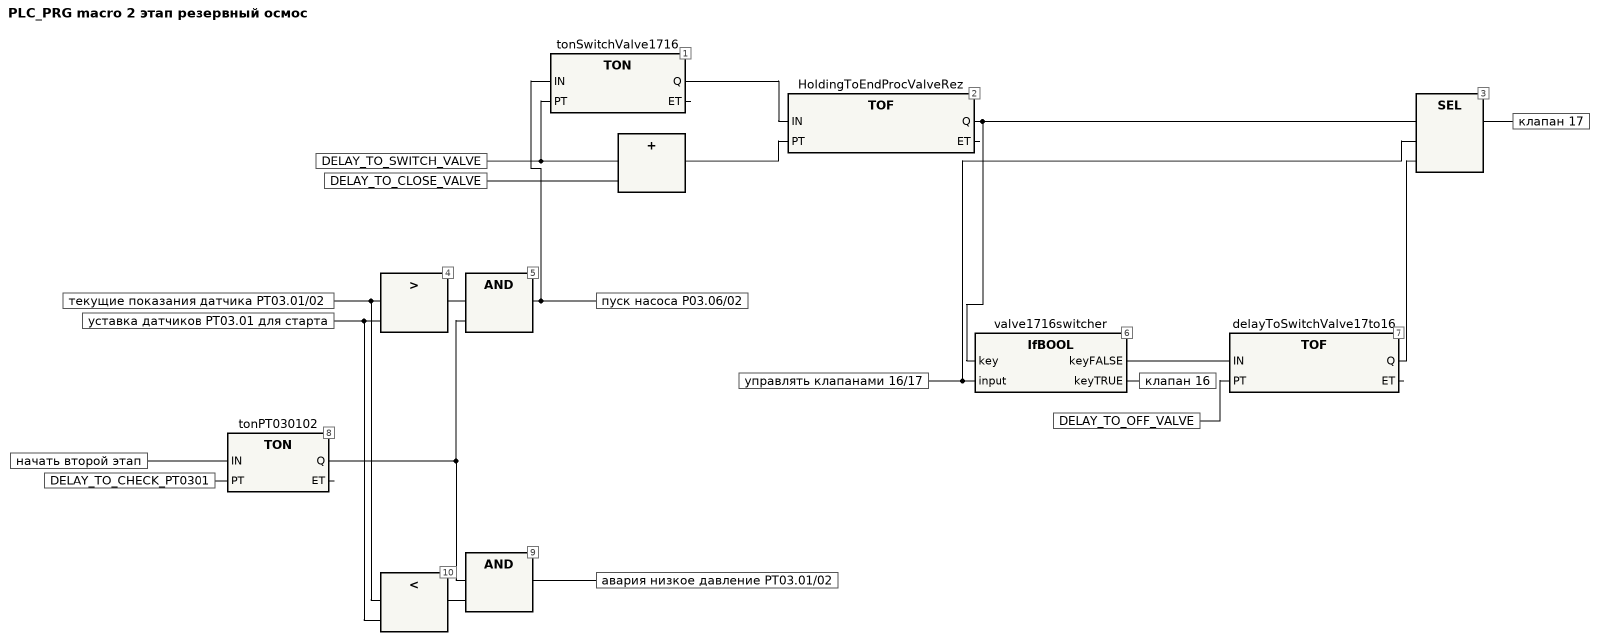
[picture p24: PLC_PRG macro 2 этап резервный осмос (CFC)]
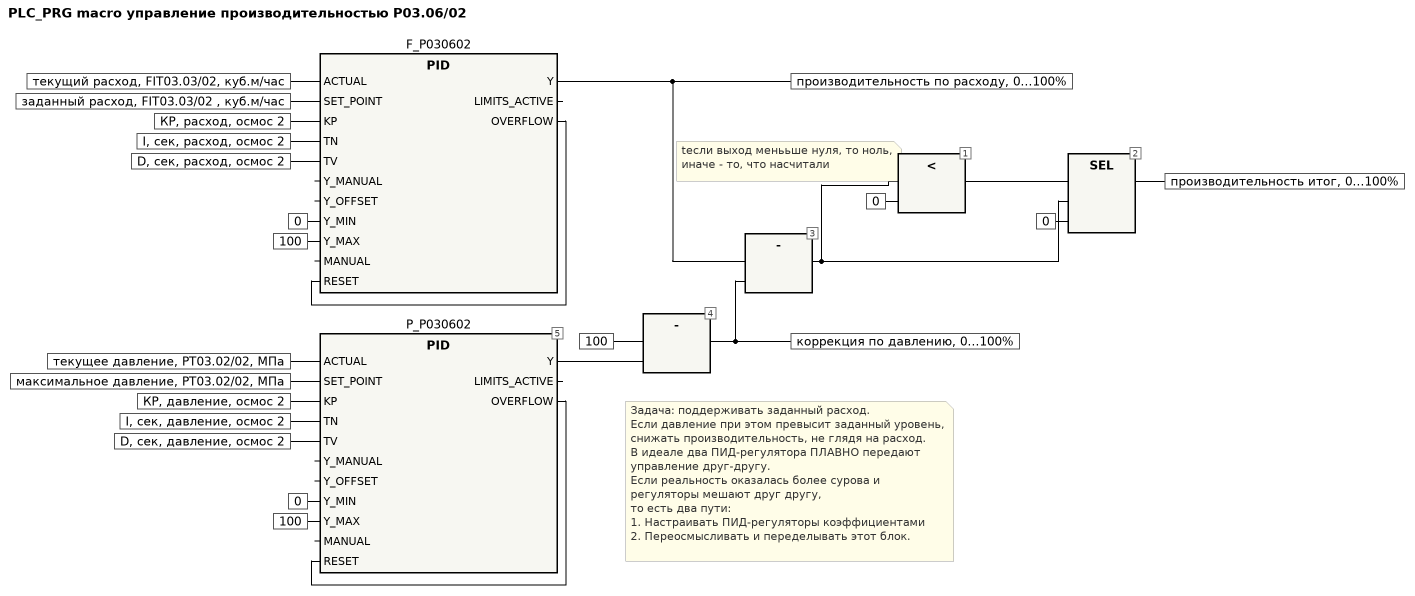
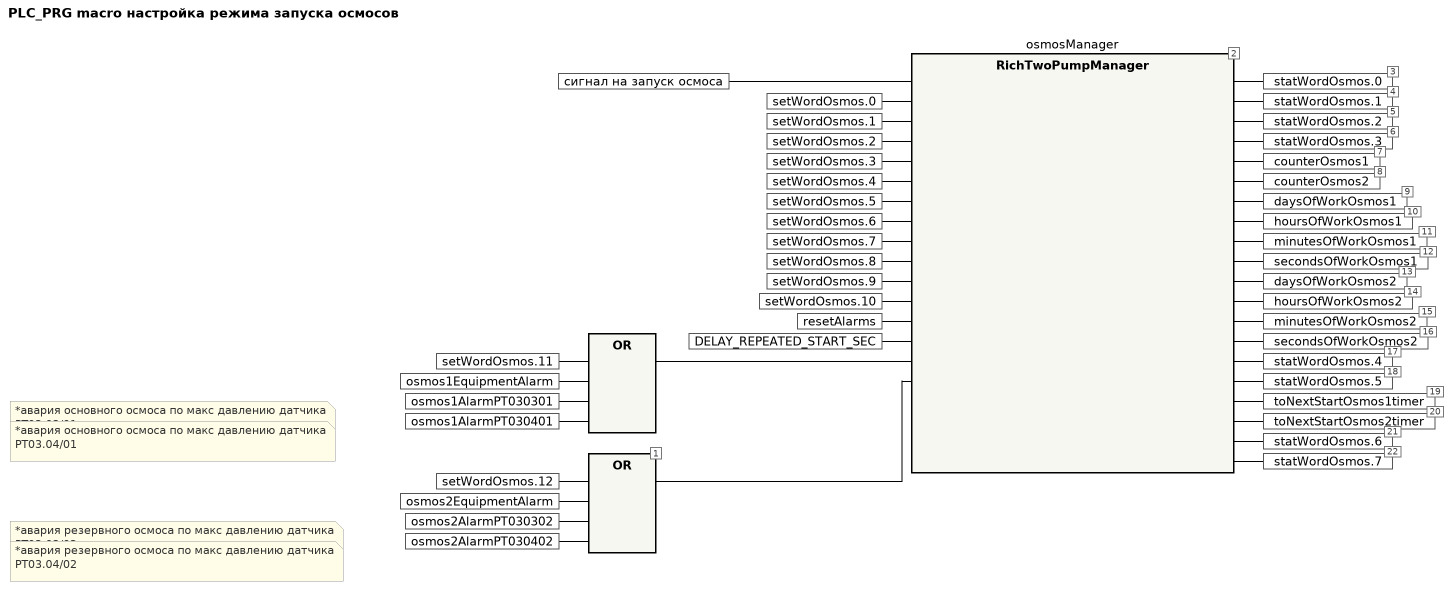
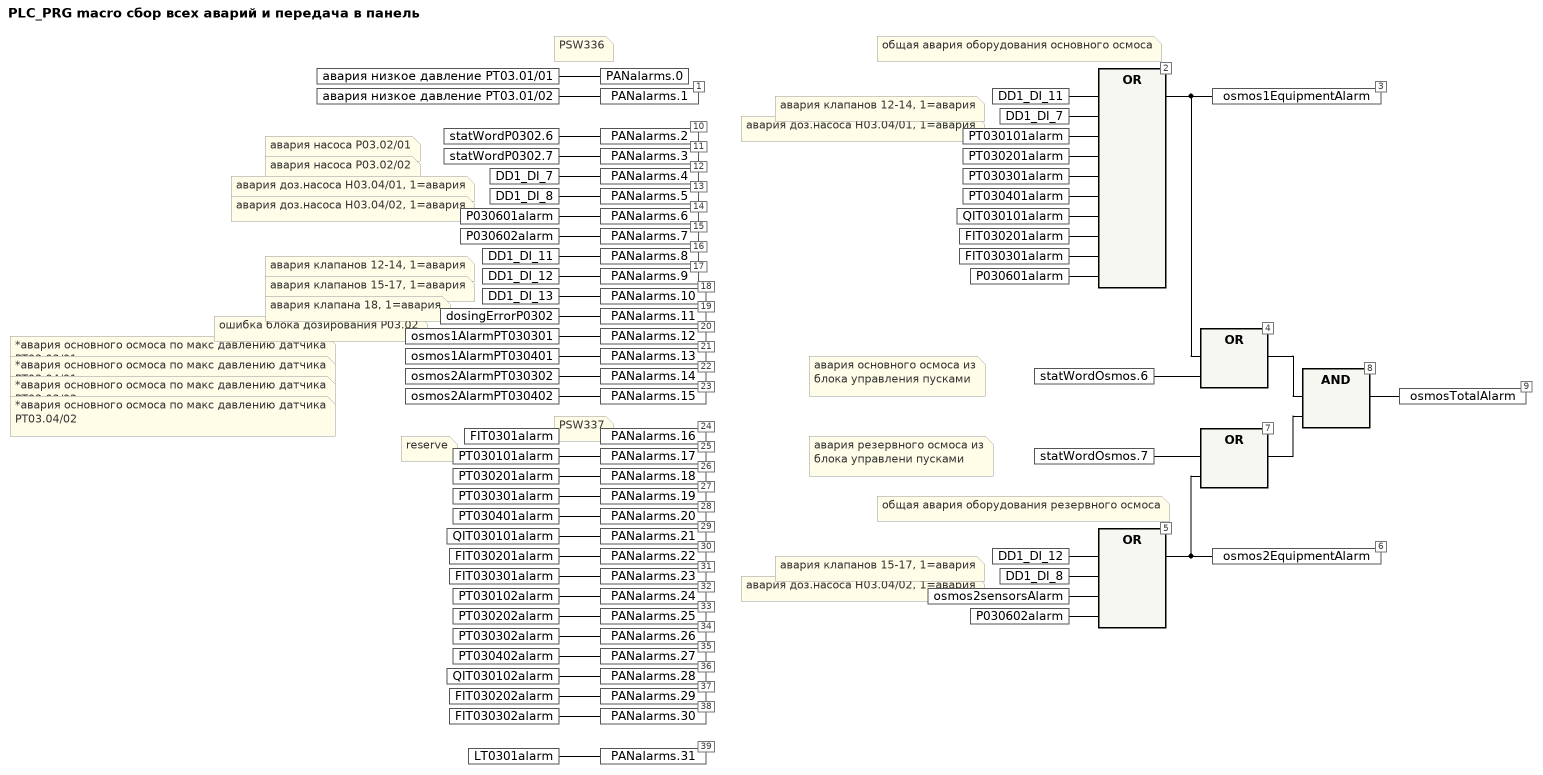
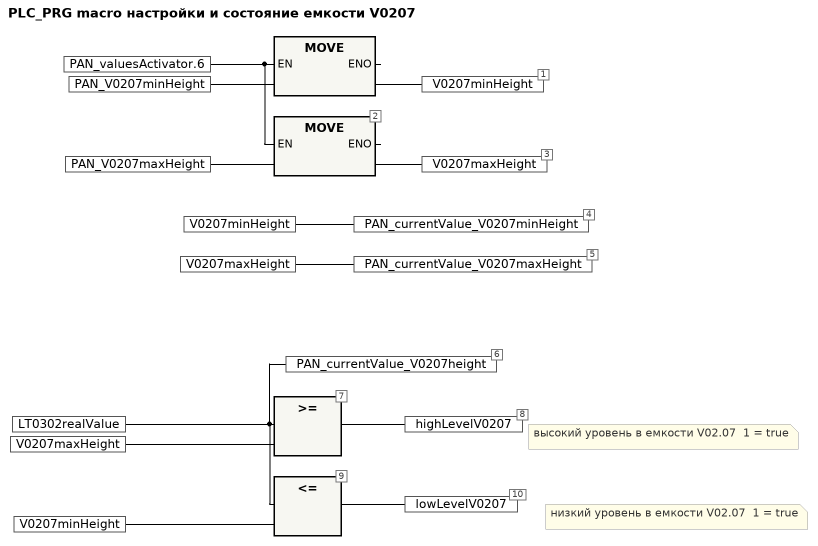
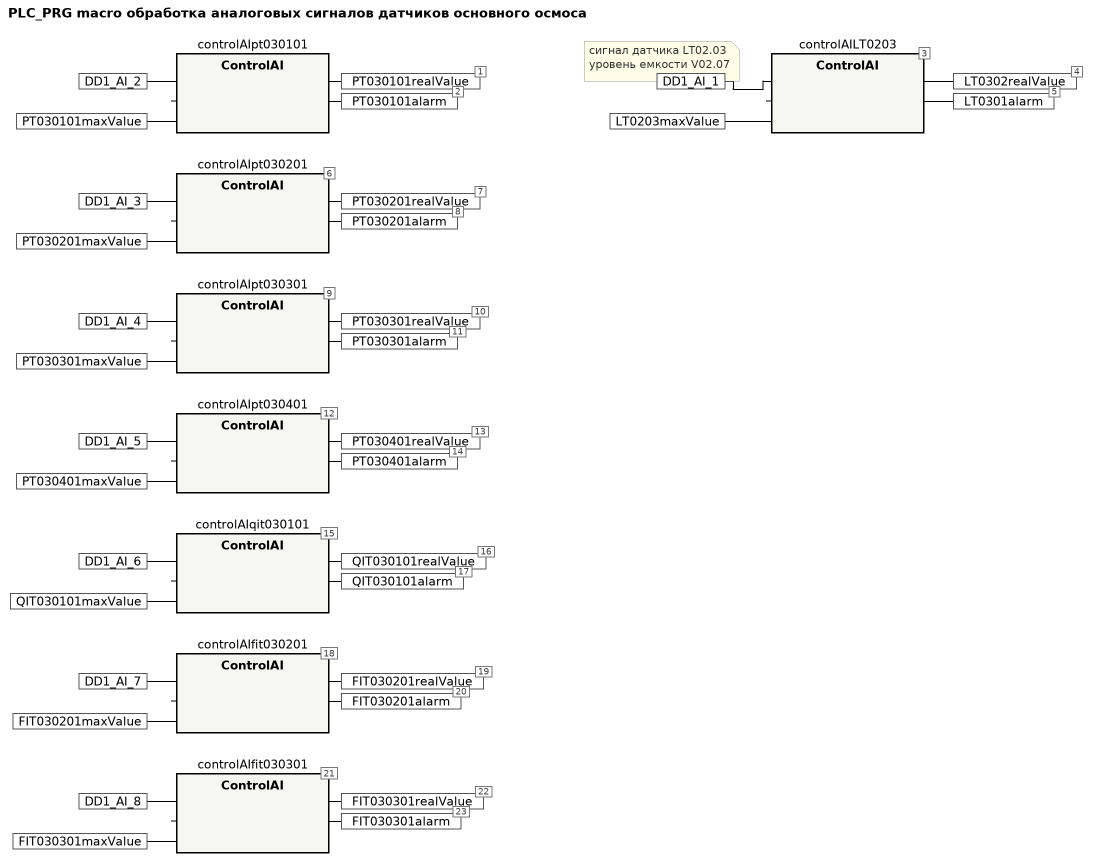
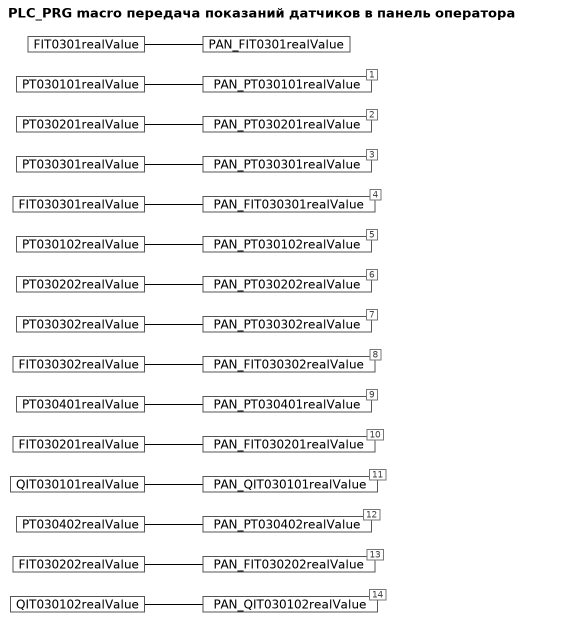
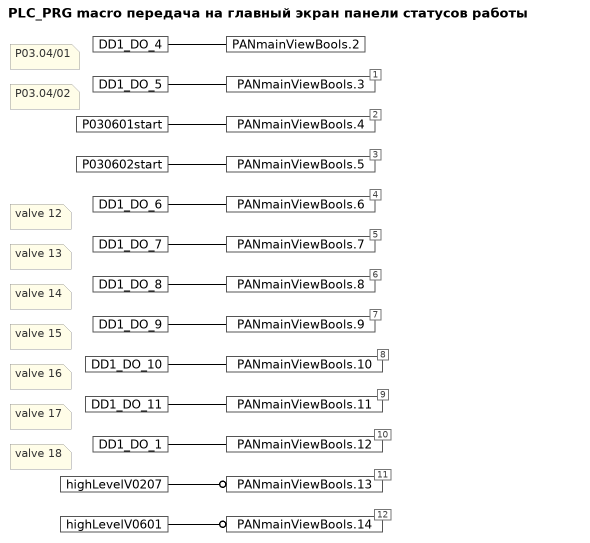
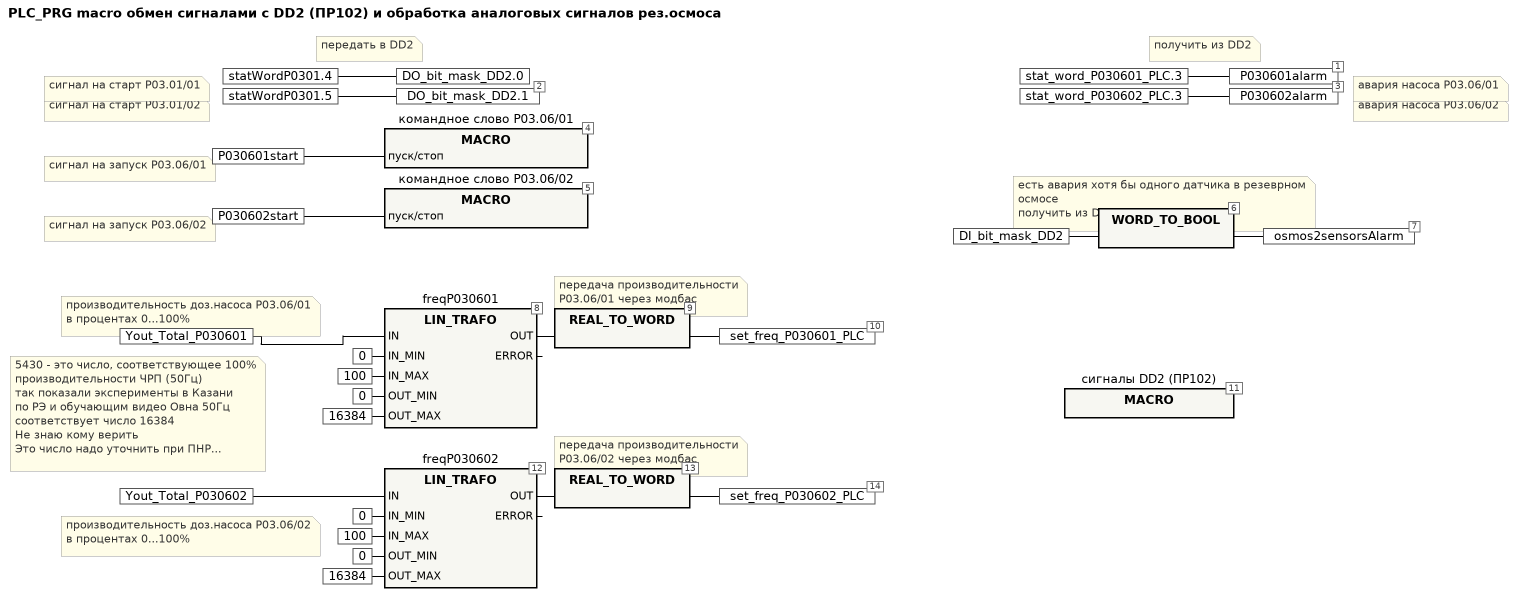
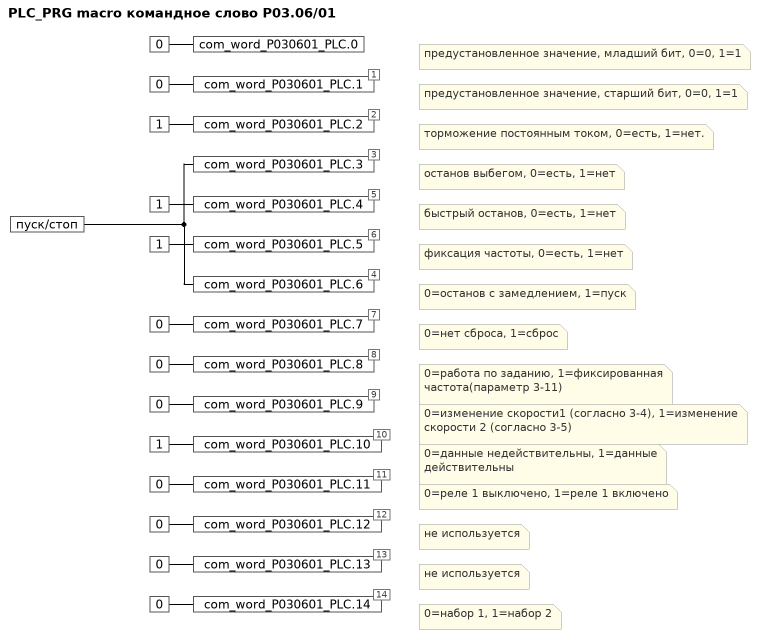
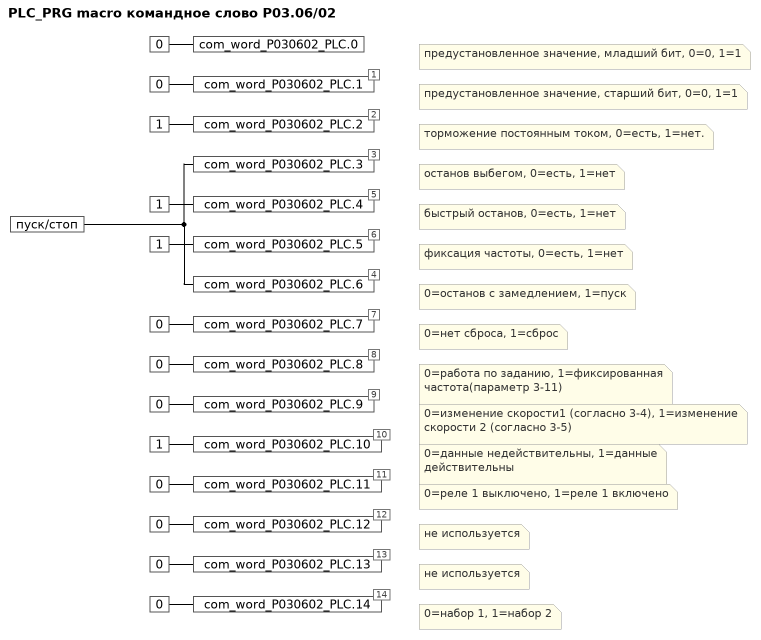
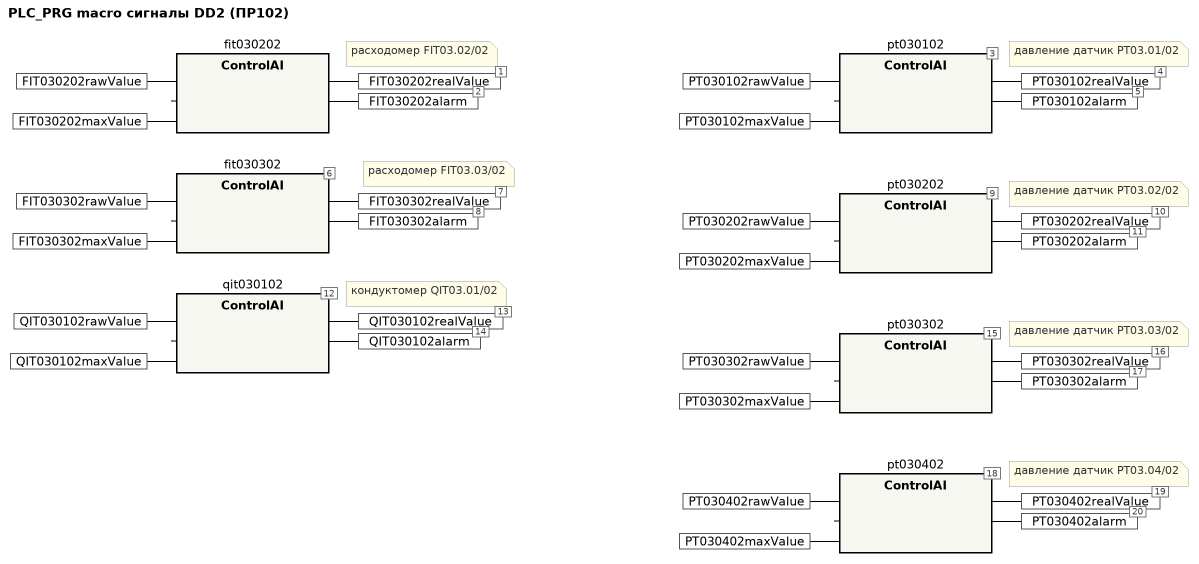
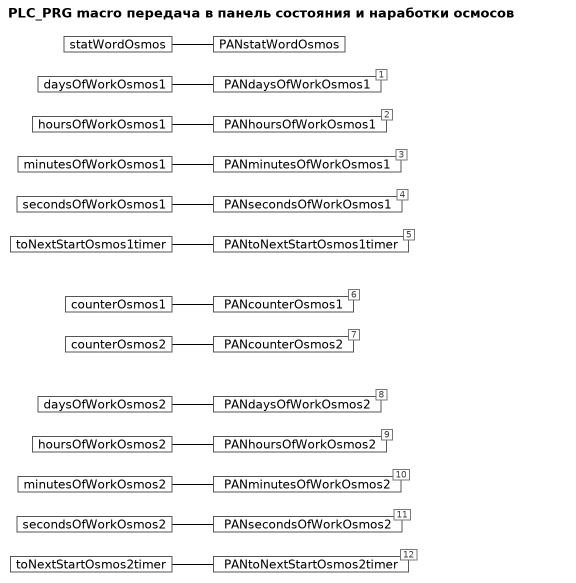
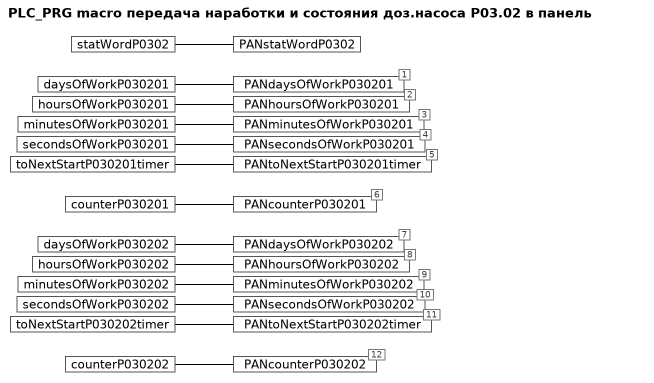
_CFC_ (* Continuous Function Chart, elements in execution order *)
(* принять сигнал из АСУ1, / FIT01.02, куб.м.час *)
(* Здесь это FIt01.02 / FIT0301 - название из алгоритма от второго осмоса *)
(* в осмосе 2 это было "Показания расходомера FIT03.01/01 на входе в осмос 2. / Для управления производительностью НД Р03.02 (1 и 2)." *)
(* пропиши в конфигурации ПЛК / ********************************** *)
(* пропиши в конфигурации ПЛК / ********************************** *)
(* авария обоих осмосов, 1 = авария *)
(* авария клапана 18, 1 = авария *)
(* авария обоих доз. насосов / Р03.02 на входе в осмос, 1 = авария *)
(* условие на запуск осмоса: / - высокий уровень в емкости V02.07 = false / - высокий уровень в емкости V06.01 = false / - высокий уровень в емкости V04.01 (БМТ) *)
(* - высокий уровень в емкости V02.07 / 1 = true *)
(* - высокий уровень в емкости V06.01 / (сигнал из АСУ-1 общий) 1 = true *)
(* алгоритм полностью скопирован из осмос-2 АСУ-3, / поэтому имена переменных многие будут оттуда, однако, в панели они / будут подписаны правильно! / Также здесь удалены насосы подачи на осмос Р03.01 / И условие запуска осмосов не такое, как в осмос-2 / Здесь запуск если V02.07  - !! нет сигнала что уровень высокий !! / (в осмос 2 - если уровень низкий) / емкость в БМТ не отслеживаем, а уровень в V06.01  условие то же / что и в осмос 2. *)
(* восстановление заданного ранее режима / работы после подачи питания *)
(* - высокий уровень в емкости V06.01 / (сигнал из АСУ-1 общий) 1 = true *)
(* расход в БМТ для расчета каскадной уставки / получить из АСУ-1! *)
(* показ расхода БМТ в панели оператора *)
(* 0 = уставка расходу своя, не каскад / 1 = уставка каскадная от расхода БМТ *)
(* прием/передача сигналов *)
(* командное слово для осмоса *)
(* командное слово доз. насоса Р03.02 *)
(* PAN - переменные для панели в щите / OPAN - переменные для выносной панели, на установке *)
(* ******************добавь сюда вкл и выкл от выносной панели******************* / задание режима работы - каскад/не каскад *)
(* передать в АСУ 1 для / передачи в осмос 2 *)
(* авария датчика уровня LT0203 *)
#0 onStartCatcher:R_TRIG(CLK: TRUE)
#1 OR(PANsetWordOsmos.11, #0.Q)
#2 resetAlarms <= #1
#3 setCascadeOnStart:IfBOOL(key: isCascadeOnStart, input: #0.Q)
#4 OR(#3.keyTRUE, PANsetWordOsmos.12)
#5 OR(#3.keyFALSE, PANsetWordOsmos.13)
#6 cascadeTrig:RS(SET: #4, RESET1: #5)
#7 statWordOsmos.8 <= #6.Q1
#8 isCascade <= #6.Q1
#9 OR(#4, #5)
#10 MOVE(EN: #9, isCascade)
#11 isCascadeOnStart <= #10
#12 MOVE(EN: #0.Q, setWordP0302onStart)
#13 setWordP0302 <= #12
#14 MOVE(EN: #0.Q, setWordOsmosOnStart)
#15 setWordOsmos <= #14
#16 ASU_Levels_output.0 <= lowLevelV0207
#17 highLevelV0601 <= ASU_Levels_input.0
#18 BMTflowToCascade <= ASU_FlowFromBMT
#19 FIT0301realValue <= ASU_FlowFIT0102
#20 MACRO алгоритм работы доз.насосов Р03.02(pin 1 "показания расходомера на входе": ASU_FlowFIT0102)
	(* приходит из макроса "алгоритм работы осмосов" *)
	(* авт.выкл и сигнал от самого / доз.насоса Р03.02/02 / 1 = норма, 0 = авария *)
	(* авт.выкл и сигнал от самого / доз.насоса Р03.02/01 / 1 = норма, 0 = авария *)
	(* Доз.насосы Р03.02/01 и Р03.02/02 на входе в осмос 2 *)
	(* выход на пуск Р03.02/01 *)
	(* задание производительности Р03.02/01 *)
	(* задание производительности Р03.02/02 *)
	(* выход на пуск Р03.02/02 *)
	(* invers alarms!!!!!!!!! *)
	#21 P0302:RichTwoPumpManager(startP0302, setWordP0302.0, setWordP0302.1, setWordP0302.2, setWordP0302.3, setWordP0302.4, setWordP0302.5, setWordP0302.6, setWordP0302.7, setWordP0302.8, setWordP0302.9, setWordP0302.10, resetAlarms, DELAY_REPEATED_START_SEC, DD1_DI_5, DD1_DI_6)
	#22 statWordP0302.0 <= #21.out 1
	#23 statWordP0302.1 <= #21.out 2
	#24 statWordP0302.2 <= #21.out 3
	#25 statWordP0302.3 <= #21.out 4
	#26 counterP030201 <= #21.out 5
	#27 counterP030202 <= #21.out 6
	#28 daysOfWorkP030201 <= #21.out 7
	#29 hoursOfWorkP030201 <= #21.out 8
	#30 minutesOfWorkP030201 <= #21.out 9
	#31 secondsOfWorkP030201 <= #21.out 10
	#32 daysOfWorkP030202 <= #21.out 11
	#33 hoursOfWorkP030202 <= #21.out 12
	#34 minutesOfWorkP030202 <= #21.out 13
	#35 secondsOfWorkP030202 <= #21.out 14
	#36 statWordP0302.4 <= #21.out 15
	#37 DD1_DO_2 <= #21.out 15
	#38 DD1_DO_3 <= #21.out 16
	#39 toNextStartP030201timer <= #21.out 17
	#40 statWordP0302.5 <= #21.out 16
	#41 toNextStartP030202timer <= #21.out 18
	#42 statWordP0302.6 <= #21.out 19
	#43 statWordP0302.7 <= #21.out 20
	#44 SEL(statWordP0302.4, 4.00, #46.out 1)
	#45 DD1_AO_1 <= #44
	#46 P0302dos:DosingPumpProportional(pin 1, -, setMaxPumpDosingValueP0302, -, -, setKoeffProportionalityP0302, -)
	#47 dosingErrorP0302 <= #46.out 2
	#48 SEL(statWordP0302.5, 4.00, #46.out 1)
	#49 DD1_AO_2 <= #48
END_MACRO
#50 MACRO настройка расхода, каскада и допустимых давлений осмоса()
	(* значение, вычитаемое из расхода БМТ / задается в панели, коэф.каскад *)
	(* предельно допустимые давления *)
	(* некаскадная уставка на поддержание расхода *)
	(* мин.давление для старта осмосов *)
	#51 MOVE(EN: PAN_valuesActivator.0, PAN_FIT0303_SetCascade)
	#52 FIT0303_SetCascade <= #51
	#53 MOVE(EN: PAN_valuesActivator.0, PAN_PT0301startValue)
	#54 PT0301startValue <= #53
	#55 MOVE(EN: PAN_valuesActivator.0, PAN_FIT0303setValue)
	#56 FIT0303setValue <= #55
	#57 MOVE(EN: PAN_valuesActivator.0, PAN_PT0302setMaxValue)
	#58 PT0302setMaxValue <= #57
	#59 MOVE(EN: PAN_valuesActivator.0, PAN_PT0303setMaxValue)
	#60 PT0303setMaxValue <= #59
	#61 MOVE(EN: PAN_valuesActivator.0, PAN_PT0304setMaxValue)
	#62 PT0304setMaxValue <= #61
	#63 PAN_currentValue_PT0301startValue <= PT0301startValue
	#64 PAN_currentValue_FIT0303setValue <= FIT0303setValue
	#65 PAN_currentValue_PT0302setMaxValue <= PT0302setMaxValue
	#66 PAN_currentValue_PT0303setMaxValue <= PT0303setMaxValue
	#67 PAN_currentValue_PT0304setMaxValue <= PT0304setMaxValue
	#68 PAN_currentValue_FIT0303_SetCascade <= FIT0303_SetCascade
END_MACRO
#69 MACRO коэффициенты ПИД-регуляторов осмосов()
	(* осмос 1 *)
	(* осмос 2 *)
	(* PID по расходу *)
	(* PID по давлению *)
	(* PID по расходу *)
	(* PID по давлению *)
	#70 MOVE(EN: PAN_valuesActivator.1, PAN_KP_F_P030601)
	#71 KP_F_P030601 <= #70
	#72 MOVE(EN: PAN_valuesActivator.1, PAN_I_F_P030601)
	#73 I_F_P030601 <= #72
	#74 MOVE(EN: PAN_valuesActivator.1, PAN_D_F_P030601)
	#75 D_F_P030601 <= #74
	#76 MOVE(EN: PAN_valuesActivator.1, PAN_KP_P_P030601)
	#77 KP_P_P030601 <= #76
	#78 MOVE(EN: PAN_valuesActivator.1, PAN_I_P_P030601)
	#79 I_P_P030601 <= #78
	#80 MOVE(EN: PAN_valuesActivator.1, PAN_D_P_P030601)
	#81 D_P_P030601 <= #80
	#82 MOVE(EN: PAN_valuesActivator.2, PAN_KP_F_P030602)
	#83 KP_F_P030602 <= #82
	#84 MOVE(EN: PAN_valuesActivator.2, PAN_I_F_P030602)
	#85 I_F_P030602 <= #84
	#86 MOVE(EN: PAN_valuesActivator.2, PAN_D_F_P030602)
	#87 D_F_P030602 <= #86
	#88 MOVE(EN: PAN_valuesActivator.2, PAN_KP_P_P030602)
	#89 KP_P_P030602 <= #88
	#90 MOVE(EN: PAN_valuesActivator.2, PAN_I_P_P030602)
	#91 I_P_P030602 <= #90
	#92 MOVE(EN: PAN_valuesActivator.2, PAN_D_P_P030602)
	#93 D_P_P030602 <= #92
	#94 PAN_currentValue_KP_F_P030601 <= KP_F_P030601
	#95 PAN_currentValue_KP_F_P030602 <= KP_F_P030602
	#96 PAN_currentValue_I_F_P030601 <= I_F_P030601
	#97 PAN_currentValue_I_F_P030602 <= I_F_P030602
	#98 PAN_currentValue_D_F_P030601 <= D_F_P030601
	#99 PAN_currentValue_D_F_P030602 <= D_F_P030602
	#100 PAN_currentValue_KP_P_P030601 <= KP_P_P030601
	#101 PAN_currentValue_KP_P_P030602 <= KP_P_P030602
	#102 PAN_currentValue_I_P_P030601 <= I_P_P030601
	#103 PAN_currentValue_I_P_P030602 <= I_P_P030602
	#104 PAN_currentValue_D_P_P030601 <= D_P_P030601
	#105 PAN_currentValue_D_P_P030602 <= D_P_P030602
END_MACRO
#106 WORD_TO_BOOL(PANsetWordP0302)
#107 tof3:TOF(IN: #106, PT: T#1s)
#108 MOVE(EN: #107.Q, PANsetWordP0302)
#109 setWordP0302 <= #108
#110 WORD_TO_BOOL(OPANsetWordP0302)
#111 tof4:TOF(IN: #110, PT: T#1s)
#112 OR(#107.Q, #111.Q)
#113 MOVE(EN: #112, statWordP0302)
#114 setWordP0302onStart <= #113
#115 MOVE(EN: #111.Q, OPANsetWordP0302)
#116 setWordP0302 <= #115
#117 MACRO уставки доз.насосов Р03.02()
	(* max производительность доз.насоса Р03.02 *)
	(* задание дозирования, мл/куб.м *)
	#118 MOVE(EN: PAN_valuesActivator.3, PANsetMaxPumpDosingValueP0302)
	#119 setMaxPumpDosingValueP0302 <= #118
	#120 MOVE(EN: PAN_valuesActivator.3, PANsetKoeffPropotrionalityP0302)
	#121 setKoeffProportionalityP0302 <= #120
	#122 PAN_currentValue_setMaxPumpDosingValueP0302 <= setMaxPumpDosingValueP0302
	#123 PAN_currentValue_setKoeffProportionalityP0302 <= setKoeffProportionalityP0302
END_MACRO
#124 PAN_BMT_Flow <= BMTflowToCascade
#125 MACRO задание задержек времени из панели()
	(* задержка до переключения клапанов после запуска Р0306 *)
	(* задержка перед открытием/закрытием клапанов при / последовательном открытии/закрытии при старте осмоса *)
	(* время задержки начала контроля параметра (например, задержка / контроля эк.манометра после насоса, время на разгон). *)
	(* Время задержки повторного пуска насосов, сек *)
	(* задержка контроля датчика РТ0301 *)
	(* задержка до начала закрытия клапанов после выключения насоса *)
	(* T#5s *)
	(* 15 *)
	(* T#3s *)
	(* T#10s *)
	(* T#15s *)
	(* T#10s *)
	#126 MACRO word to time(pin 1 "word_in": PAN_CHECKING_DELAY_TIME)
		#127 UINT_TO_UDINT(pin 1)
		#128 MUL(#127, 1000)
		#129 UDINT_TO_TIME(#128)
		out 1 "time_out" <= #129
	END_MACRO
	#130 MOVE(EN: PAN_valuesActivator.4, #126.out 1)
	#131 CHECKING_DELAY_TIME <= #130
	#132 MOVE(EN: PAN_valuesActivator.4, PAN_DELAY_REPEATED_START_SEC)
	#133 DELAY_REPEATED_START_SEC <= #132
	#134 MACRO word to time(pin 1 "word_in": PAN_DELAY_TO_OFF_VALVE)
		#135 UINT_TO_UDINT(pin 1)
		#136 MUL(#135, 1000)
		#137 UDINT_TO_TIME(#136)
		out 1 "time_out" <= #137
	END_MACRO
	#138 MOVE(EN: PAN_valuesActivator.4, #134.out 1)
	#139 DELAY_TO_OFF_VALVE <= #138
	#140 MACRO word to time(pin 1 "word_in": PAN_DELAY_TO_CHECK_PT0301)
		#141 UINT_TO_UDINT(pin 1)
		#142 MUL(#141, 1000)
		#143 UDINT_TO_TIME(#142)
		out 1 "time_out" <= #143
	END_MACRO
	#144 MOVE(EN: PAN_valuesActivator.4, #140.out 1)
	#145 DELAY_TO_CHECK_PT0301 <= #144
	#146 MACRO word to time(pin 1 "word_in": PAN_DELAY_TO_SWITCH_VALVE)
		#147 UINT_TO_UDINT(pin 1)
		#148 MUL(#147, 1000)
		#149 UDINT_TO_TIME(#148)
		out 1 "time_out" <= #149
	END_MACRO
	#150 MOVE(EN: PAN_valuesActivator.4, #146.out 1)
	#151 DELAY_TO_SWITCH_VALVE <= #150
	#152 MACRO word to time(pin 1 "word_in": PAN_DELAY_TO_CLOSE_VALVE)
		#153 UINT_TO_UDINT(pin 1)
		#154 MUL(#153, 1000)
		#155 UDINT_TO_TIME(#154)
		out 1 "time_out" <= #155
	END_MACRO
	#156 MOVE(EN: PAN_valuesActivator.4, #152.out 1)
	#157 DELAY_TO_CLOSE_VALVE <= #156
	#158 MACRO time to word(pin 1 "time_in": CHECKING_DELAY_TIME)
		#159 TIME_TO_UDINT(pin 1)
		#160 DIV(#159, 1000)
		#161 UDINT_TO_UINT(#160)
		out 1 "uint_out" <= #161
	END_MACRO
	#162 PAN_currentValue_CHECKING_DELAY_TIME <= #158.out 1
	#163 PAN_currentValue_DELAY_REPEATED_START_SEC <= DELAY_REPEATED_START_SEC
	#164 MACRO time to word(pin 1 "time_in": DELAY_TO_OFF_VALVE)
		#165 TIME_TO_UDINT(pin 1)
		#166 DIV(#165, 1000)
		#167 UDINT_TO_UINT(#166)
		out 1 "uint_out" <= #167
	END_MACRO
	#168 PAN_currentValue_DELAY_TO_OFF_VALVE <= #164.out 1
	#169 MACRO time to word(pin 1 "time_in": DELAY_TO_CHECK_PT0301)
		#170 TIME_TO_UDINT(pin 1)
		#171 DIV(#170, 1000)
		#172 UDINT_TO_UINT(#171)
		out 1 "uint_out" <= #172
	END_MACRO
	#173 PAN_currentValue_DELAY_TO_CHECK_PT0301 <= #169.out 1
	#174 MACRO time to word(pin 1 "time_in": DELAY_TO_SWITCH_VALVE)
		#175 TIME_TO_UDINT(pin 1)
		#176 DIV(#175, 1000)
		#177 UDINT_TO_UINT(#176)
		out 1 "uint_out" <= #177
	END_MACRO
	#178 PAN_currentValue_DELAY_TO_SWITCH_VALVE <= #174.out 1
	#179 MACRO time to word(pin 1 "time_in": DELAY_TO_CLOSE_VALVE)
		#180 TIME_TO_UDINT(pin 1)
		#181 DIV(#180, 1000)
		#182 UDINT_TO_UINT(#181)
		out 1 "uint_out" <= #182
	END_MACRO
	#183 PAN_currentValue_DELAY_TO_CLOSE_VALVE <= #179.out 1
END_MACRO
#184 MACRO настройка датчиков()
	#185 MOVE(EN: PAN_valuesActivator.5, PAN_PT030101maxValue)
	#186 PT030101maxValue <= #185
	#187 MOVE(EN: PAN_valuesActivator.5, PAN_FIT030201maxValue)
	#188 FIT030201maxValue <= #187
	#189 MOVE(EN: PAN_valuesActivator.5, PAN_PT030201maxValue)
	#190 PT030201maxValue <= #189
	#191 MOVE(EN: PAN_valuesActivator.5, PAN_FIT030301maxValue)
	#192 FIT030301maxValue <= #191
	#193 MOVE(EN: PAN_valuesActivator.5, PAN_PT030301maxValue)
	#194 PT030301maxValue <= #193
	#195 MOVE(EN: PAN_valuesActivator.5, PAN_FIT030202maxValue)
	#196 FIT030202maxValue <= #195
	#197 MOVE(EN: PAN_valuesActivator.5, PAN_PT030401maxValue)
	#198 PT030401maxValue <= #197
	#199 MOVE(EN: PAN_valuesActivator.5, PAN_FIT030302maxValue)
	#200 FIT030302maxValue <= #199
	#201 MOVE(EN: PAN_valuesActivator.5, PAN_PT030102maxValue)
	#202 PT030102maxValue <= #201
	#203 MOVE(EN: PAN_valuesActivator.5, PAN_QIT030101maxValue)
	#204 QIT030101maxValue <= #203
	#205 MOVE(EN: PAN_valuesActivator.5, PAN_PT030202maxValue)
	#206 PT030202maxValue <= #205
	#207 MOVE(EN: PAN_valuesActivator.5, PAN_QIT030102maxValue)
	#208 QIT030102maxValue <= #207
	#209 MOVE(EN: PAN_valuesActivator.5, PAN_PT030302maxValue)
	#210 PT030302maxValue <= #209
	#211 MOVE(EN: PAN_valuesActivator.5, PAN_LT0203maxValue)
	#212 LT0203maxValue <= #211
	#213 MOVE(EN: PAN_valuesActivator.5, PAN_PT030402maxValue)
	#214 PT030402maxValue <= #213
	#215 PAN_currentValue_FIT0301maxValue <= FIT0301maxValue
	#216 PAN_currentValue_PT030101maxValue <= PT030101maxValue
	#217 PAN_currentValue_FIT030201maxValue <= FIT030201maxValue
	#218 PAN_currentValue_PT030201maxValue <= PT030201maxValue
	#219 PAN_currentValue_FIT030301maxValue <= FIT030301maxValue
	#220 PAN_currentValue_PT030301maxValue <= PT030301maxValue
	#221 PAN_currentValue_FIT030202maxValue <= FIT030202maxValue
	#222 PAN_currentValue_PT030401maxValue <= PT030401maxValue
	#223 PAN_currentValue_FIT030302maxValue <= FIT030302maxValue
	#224 PAN_currentValue_PT030102maxValue <= PT030102maxValue
	#225 PAN_currentValue_QIT030101maxValue <= QIT030101maxValue
	#226 PAN_currentValue_PT030202maxValue <= PT030202maxValue
	#227 PAN_currentValue_QIT030102maxValue <= QIT030102maxValue
	#228 PAN_currentValue_PT030302maxValue <= PT030302maxValue
	#229 PAN_currentValue_PT030402maxValue <= PT030402maxValue
	#230 PAN_currentValue_LT0203maxValue <= LT0203maxValue
END_MACRO
#231 MACRO алгоритм работы осмосов (насосы Р03.06)()
	(* старт НД03.04/01 *)
	(* пуск основного осмоса *)
	(* клапан 12 *)
	(* клапан 14 *)
	(* клапан 13 *)
	(* клапан 18 *)
	(* старт НД03.04/02 *)
	(* пуск резервного осмоса *)
	(* клапан 15 *)
	(* клапан 17 *)
	(* клапан 16 *)
	(* 0 = уставка расходу своя, не каскад / 1 = уставка каскадная от расхода БМТ *)
	#232 SUB(BMTflowToCascade, FIT0303_SetCascade)
	#233 SEL(isCascade, FIT0303setValue, #232)
	#234 MACRO основной осмос(pin 1 "пуск основного осмоса": statWordOsmos.4, pin 2 "текущие показания датчика РТ03.01/01, МПа": PT030101realValue, pin 3 "уставка датчиков РТ03.01 для старта, МПа": PT0301startValue, pin 4 "текущий расход FIT03,03/01, куб.м/час": FIT030301realValue, pin 5 "заданный расход FIT03,03/01, куб.м/час": #233, pin 6 "КР, расход осн.осм.": KP_F_P030601, pin 7 "I, расход осн.осм.": I_F_P030601, pin 8 "D, расход осн.осм.": D_F_P030601, pin 9 "текущее давление, РТ03.02/01, МПа": PT030201realValue, pin 10 "максимальное давление, РТ03.02/01, МПа": PT0302setMaxValue, pin 11 "КР, давление осн.осм.": KP_P_P030601, pin 12 "I, давление осн.осм.": I_P_P030601, pin 13 "D, давление осн.осм.": D_P_P030601, pin 14 "текущие показания датчика РТ03.03/01, МПа": PT030301realValue, pin 15 "уставка max давление РТ03.03, МПа": PT0303setMaxValue, pin 16 "текущие показания датчика РТ03.04/01, МПа": PT030401realValue, pin 17 "уставка max давление РТ03.04, МПа": PT0304setMaxValue)
		#235 MACRO 1 этап основной осмос(pin 1 "пуск основного осмоса": pin 1)
			#236 OR(pin 1, #243.Q)
			out 2 "клапан 12" <= #236
			#237 tonValve14:TON(IN: pin 1, PT: DELAY_TO_OFF_VALVE)
			#238 OR(#237.Q, #242.Q)
			out 1 "клапан 14/13" <= #238
			out 3 "старт НД03.04/01" <= #239.Q
			out 5 "startP0302" <= #239.Q
			#239 tonValve18:TON(IN: #237.Q, PT: DELAY_TO_OFF_VALVE)
			#240 OR(#239.Q, #241.Q)
			out 4 "клапан 18" <= #240
			#241 tofValve18:TOF(IN: #239.Q, PT: DELAY_TO_CLOSE_VALVE)
			#242 tofValve14:TOF(IN: #241.Q, PT: DELAY_TO_OFF_VALVE)
			#243 tofValve12:TOF(IN: #242.Q, PT: DELAY_TO_OFF_VALVE)
		END_MACRO
		out 7 "клапан 12" <= #235.out 2
		out 11 "старт НД03.04/01" <= #235.out 3
		out 10 "клапан 18" <= #235.out 4
		out 12 "старт доз.насосов Р03.02" <= #235.out 5
		#244 MACRO 2 этап основной осмос(pin 1 "управлять клапанами 13/14": #235.out 1, pin 2 "начать второй этап": #235.out 5, pin 3 "текущие показания датчика РТ03.01/01": pin 2, pin 4 "уставка датчиков РТ03.01 для старта": pin 3)
			#245 +(DELAY_TO_SWITCH_VALVE, DELAY_TO_CLOSE_VALVE)
			#246 tonSwitchValve1413:TON(IN: #250, PT: DELAY_TO_SWITCH_VALVE)
			#247 HoldingToEndProcValve:TOF(IN: #246.Q, PT: #245)
			#248 SEL(#247.Q, pin 1, #252.Q)
			out 1 "клапан 14" <= #248
			#249 >(pin 3, pin 4)
			#250 AND(#249, #253.Q)
			out 4 "пуск насоса Р03.06/01" <= #250
			#251 valve1413switcher:IfBOOL(key: #247.Q, input: pin 1)
			#252 delayToSwitchValve14to13:TOF(IN: #251.keyFALSE, PT: DELAY_TO_OFF_VALVE)
			out 2 "клапан 13" <= #251.keyTRUE
			#253 tonPT030101:TON(IN: pin 2, PT: DELAY_TO_CHECK_PT0301)
			#254 AND(#253.Q, #255)
			out 3 "авария низкое давление РТ03.01/01" <= #254
			#255 <(pin 3, pin 4)
		END_MACRO
		out 9 "клапан 14" <= #244.out 1
		out 8 "клапан 13" <= #244.out 2
		out 13 "авария низкое давление РТ03.01/01" <= #244.out 3
		out 1 "пуск насоса Р03.06/01" <= #244.out 4
		#256 AND(#244.out 4, #257)
		out 2 "авария осмос 1  макс.давл.РТ03.03/01" <= #256
		#257 >=(pin 14, pin 15)
		#258 AND(#244.out 4, #259)
		out 3 "авария осмос 1  макс.давл.РТ03.04/01" <= #258
		#259 >=(pin 16, pin 17)
		#260 MACRO управление производительностью Р03.06/01(pin 1 "текущий расход, FIT03.03/01, куб.м/час": pin 4, pin 2 "заданный расход, FIT03.03/01 , куб.м/час": pin 5, pin 3 "КР, расход": pin 6, pin 4 "I, сек, расход": pin 7, pin 5 "D, сек, расход": pin 8, pin 6 "текущее давление, РТ03.02/01, МПа": pin 9, pin 7 "максимальное давление, РТ03.02/01, МПа": pin 10, pin 8 "КР, давление": pin 11, pin 9 "I, сек, давление": pin 12, pin 10 "D, сек, давление": pin 13)
			(* Задача: поддерживать заданный расход. / Если давление при этом превысит заданный уровень, / снижать производительность, не глядя на расход. / В идеале два ПИД-регулятора ПЛАВНО передают управление друг-другу. / Если реальность оказалась более сурова и регуляторы мешают друг другу, / то есть два пути: / 1. Настраивать ПИД-регуляторы коэффициентами / 2. Переосмысливать и переделывать этот блок. *)
			(* tесли выход менььше нуля, то ноль, / иначе - то, что насчитали *)
			#261 F_P030601:PID(ACTUAL: pin 1, SET_POINT: pin 2, KP: pin 3, TN: pin 4, TV: pin 5, Y_MANUAL: -, Y_OFFSET: -, Y_MIN: 0, Y_MAX: 100, MANUAL: -, RESET: #261.OVERFLOW)
			out 1 "производительность по расходу, 0...100%" <= #261.Y
			#262 <(#264, 0)
			#263 SEL(#262, #264, 0)
			out 3 "производительность итог, 0...100%" <= #263
			#264 -(#261.Y, #265)
			#265 -(100, #266.Y)
			out 2 "коррекция по давлению, 0...100%" <= #265
			#266 P_P030601:PID(ACTUAL: pin 6, SET_POINT: pin 7, KP: pin 8, TN: pin 9, TV: pin 10, Y_MANUAL: -, Y_OFFSET: -, Y_MIN: 0, Y_MAX: 100, MANUAL: -, RESET: #266.OVERFLOW)
		END_MACRO
		out 4 "производительность по расходу осн.осмос, 0...100%" <= #260.out 1
		out 5 "коррекция по давлению осн.осмос, 0...100%" <= #260.out 2
		out 6 "производительность итог осн.осмос, 0...100%" <= #260.out 3
	END_MACRO
	#267 P030601start <= #234.out 1
	#268 osmos1AlarmPT030301 <= #234.out 2
	#269 osmos1AlarmPT030401 <= #234.out 3
	#270 Yout_F_P030601 <= #234.out 4
	#271 Yout_P_P030601 <= #234.out 5
	#272 Yout_Total_P030601 <= #234.out 6
	#273 DD1_DO_6 <= #234.out 7
	#274 DD1_DO_7 <= #234.out 8
	#275 DD1_DO_8 <= #234.out 9
	#276 DD1_DO_4 <= #234.out 11
	#277 MACRO резервный осмос(pin 1 "пуск резервного осмоса": statWordOsmos.5, pin 2 "текущие показания РТ01.03/02": PT030102realValue, pin 3 "уставка РТ03.01/02 для старта": PT0301startValue, pin 4 "текущий расход, FIT03/03/02, куб.м/час": FIT030302realValue, pin 5 "заданный расход, FIT03/03/02, куб.м/час": #233, pin 6 "KP, расход, осмос 2": KP_F_P030602, pin 7 "I, расход, осмос 2": I_F_P030602, pin 8 "D, расход, осмос 2": D_F_P030602, pin 9 "текущее давление PT03.02/02, МПа": PT030202realValue, pin 10 "максимальное давление PT03.02/02, МПа": PT0302setMaxValue, pin 11 "KP, давление, осмос 2": KP_P_P030602, pin 12 "I, давление, осмос 2": I_P_P030602, pin 13 "D, давление, осмос 2": D_P_P030602, pin 14 "текущее давление РТ03.03/02": PT030302realValue, pin 15 "задание max давление РТ03.03/02": PT0303setMaxValue, pin 16 "текущее давление РТ03.04/02": PT030402realValue, pin 17 "задание max давление РТ03.04/02": PT0304setMaxValue)
		#278 MACRO 1 этап резервный осмос(pin 1 "пуск резервного осмоса": pin 1)
			#279 OR(pin 1, #286.Q)
			out 2 "клапан 15" <= #279
			#280 tonValve17:TON(IN: pin 1, PT: DELAY_TO_OFF_VALVE)
			#281 OR(#280.Q, #285.Q)
			out 1 "клапан 16/17" <= #281
			out 3 "старт НД03.04/02" <= #282.Q
			out 5 "startP0302" <= #282.Q
			#282 tonValve18rez:TON(IN: #280.Q, PT: DELAY_TO_OFF_VALVE)
			#283 OR(#282.Q, #284.Q)
			out 4 "клапан 18" <= #283
			#284 tofValve18rez:TOF(IN: #282.Q, PT: DELAY_TO_CLOSE_VALVE)
			#285 tofValve17:TOF(IN: #284.Q, PT: DELAY_TO_OFF_VALVE)
			#286 tofValve15:TOF(IN: #285.Q, PT: DELAY_TO_OFF_VALVE)
		END_MACRO
		out 5 "клапан 15" <= #278.out 2
		out 6 "старт НД03.04/02" <= #278.out 3
		out 2 "клапан 18" <= #278.out 4
		out 1 "пуск Р0302" <= #278.out 5
		#287 MACRO 2 этап резервный осмос(pin 1 "управлять клапанами 16/17": #278.out 1, pin 2 "начать второй этап": #278.out 5, pin 3 "текущие показания датчика РТ03.01/02": pin 2, pin 4 "уставка датчиков РТ03.01 для старта": pin 3)
			#288 +(DELAY_TO_SWITCH_VALVE, DELAY_TO_CLOSE_VALVE)
			#289 tonSwitchValve1716:TON(IN: #293, PT: DELAY_TO_SWITCH_VALVE)
			#290 HoldingToEndProcValveRez:TOF(IN: #289.Q, PT: #288)
			#291 SEL(#290.Q, pin 1, #295.Q)
			out 1 "клапан 17" <= #291
			#292 >(pin 3, pin 4)
			#293 AND(#292, #296.Q)
			out 4 "пуск насоса Р03.06/02" <= #293
			#294 valve1716switcher:IfBOOL(key: #290.Q, input: pin 1)
			#295 delayToSwitchValve17to16:TOF(IN: #294.keyFALSE, PT: DELAY_TO_OFF_VALVE)
			out 2 "клапан 16" <= #294.keyTRUE
			#296 tonPT030102:TON(IN: pin 2, PT: DELAY_TO_CHECK_PT0301)
			#297 AND(#296.Q, #298)
			out 3 "авария низкое давление РТ03.01/02" <= #297
			#298 <(pin 3, pin 4)
		END_MACRO
		out 3 "клапан 17" <= #287.out 1
		out 4 "клапан 16" <= #287.out 2
		out 7 "авария низкое давление РТ03.01/02" <= #287.out 3
		out 8 "пуск насоса Р03.06/02" <= #287.out 4
		#299 AND(#287.out 4, #300)
		out 12 "авария осмос 2 max давление РТ03.03/02" <= #299
		#300 >=(pin 14, pin 15)
		#301 AND(#287.out 4, #302)
		out 13 "авария осмос 2 max давление РТ03.04/02" <= #301
		#302 >=(pin 16, pin 17)
		#303 MACRO управление производительностью Р03.06/02(pin 1 "текущий расход, FIT03.03/02, куб.м/час": pin 4, pin 2 "заданный расход, FIT03.03/02 , куб.м/час": pin 5, pin 3 "КР, расход, осмос 2": pin 6, pin 4 "I, сек, расход, осмос 2": pin 7, pin 5 "D, сек, расход, осмос 2": pin 8, pin 6 "текущее давление, РТ03.02/02, МПа": pin 9, pin 7 "максимальное давление, РТ03.02/02, МПа": pin 10, pin 8 "КР, давление, осмос 2": pin 11, pin 9 "I, сек, давление, осмос 2": pin 12, pin 10 "D, сек, давление, осмос 2": pin 13)
			(* Задача: поддерживать заданный расход. / Если давление при этом превысит заданный уровень, / снижать производительность, не глядя на расход. / В идеале два ПИД-регулятора ПЛАВНО передают управление друг-другу. / Если реальность оказалась более сурова и регуляторы мешают друг другу, / то есть два пути: / 1. Настраивать ПИД-регуляторы коэффициентами / 2. Переосмысливать и переделывать этот блок. *)
			(* tесли выход менььше нуля, то ноль, / иначе - то, что насчитали *)
			#304 F_P030602:PID(ACTUAL: pin 1, SET_POINT: pin 2, KP: pin 3, TN: pin 4, TV: pin 5, Y_MANUAL: -, Y_OFFSET: -, Y_MIN: 0, Y_MAX: 100, MANUAL: -, RESET: #304.OVERFLOW)
			out 1 "производительность по расходу, 0...100%" <= #304.Y
			#305 <(#307, 0)
			#306 SEL(#305, #307, 0)
			out 3 "производительность итог, 0...100%" <= #306
			#307 -(#304.Y, #308)
			#308 -(100, #309.Y)
			out 2 "коррекция по давлению, 0...100%" <= #308
			#309 P_P030602:PID(ACTUAL: pin 6, SET_POINT: pin 7, KP: pin 8, TN: pin 9, TV: pin 10, Y_MANUAL: -, Y_OFFSET: -, Y_MIN: 0, Y_MAX: 100, MANUAL: -, RESET: #309.OVERFLOW)
		END_MACRO
		out 9 "производительность по расходу, рез.осмос, 0...100%" <= #303.out 1
		out 10 "коррекция по давлению, рез.осмос, 0...100%" <= #303.out 2
		out 11 "производительность итог, 0...100%" <= #303.out 3
	END_MACRO
	#310 DD1_DO_11 <= #277.out 3
	#311 DD1_DO_10 <= #277.out 4
	#312 DD1_DO_9 <= #277.out 5
	#313 DD1_DO_5 <= #277.out 6
	#314 P030602start <= #277.out 8
	#315 Yout_F_P030602 <= #277.out 9
	#316 Yout_P_P030602 <= #277.out 10
	#317 Yout_Total_P030602 <= #277.out 11
	#318 osmos2AlarmPT030302 <= #277.out 12
	#319 osmos2AlarmPT030402 <= #277.out 13
	#320 OR(#234.out 10, #277.out 2)
	#321 DD1_DO_1 <= #320
	#322 OR(#234.out 12, #277.out 1)
	#323 startP0302 <= #322
	out 1 "авария низкое давление РТ03.01/01" <= #234.out 13
	out 2 "авария низкое давление РТ03.01/02" <= #277.out 7
END_MACRO
#324 AND(NOT highLevelV0207, NOT highLevelV0601)
#325 AND(NOT alarmP0302, NOT DD1_DI_13, NOT osmosTotalAlarm, NOT LT0301alarm, NOT #231.out 1, NOT #231.out 2)
#326 AND(#324, #325)
#327 MACRO настройка режима запуска осмосов(pin 1 "сигнал на запуск осмоса": #326)
	(* *авария основного осмоса по макс давлению датчика РТ03.03/01 *)
	(* *авария основного осмоса по макс давлению датчика РТ03.04/01 *)
	(* *авария резервного осмоса по макс давлению датчика РТ03.03/02 *)
	(* *авария резервного осмоса по макс давлению датчика РТ03.04/02 *)
	#328 OR(setWordOsmos.11, osmos1EquipmentAlarm, osmos1AlarmPT030301, osmos1AlarmPT030401)
	#329 OR(setWordOsmos.12, osmos2EquipmentAlarm, osmos2AlarmPT030302, osmos2AlarmPT030402)
	#330 osmosManager:RichTwoPumpManager(pin 1, setWordOsmos.0, setWordOsmos.1, setWordOsmos.2, setWordOsmos.3, setWordOsmos.4, setWordOsmos.5, setWordOsmos.6, setWordOsmos.7, setWordOsmos.8, setWordOsmos.9, setWordOsmos.10, resetAlarms, DELAY_REPEATED_START_SEC, #328, #329)
	#331 statWordOsmos.0 <= #330.out 1
	#332 statWordOsmos.1 <= #330.out 2
	#333 statWordOsmos.2 <= #330.out 3
	#334 statWordOsmos.3 <= #330.out 4
	#335 counterOsmos1 <= #330.out 5
	#336 counterOsmos2 <= #330.out 6
	#337 daysOfWorkOsmos1 <= #330.out 7
	#338 hoursOfWorkOsmos1 <= #330.out 8
	#339 minutesOfWorkOsmos1 <= #330.out 9
	#340 secondsOfWorkOsmos1 <= #330.out 10
	#341 daysOfWorkOsmos2 <= #330.out 11
	#342 hoursOfWorkOsmos2 <= #330.out 12
	#343 minutesOfWorkOsmos2 <= #330.out 13
	#344 secondsOfWorkOsmos2 <= #330.out 14
	#345 statWordOsmos.4 <= #330.out 15
	#346 statWordOsmos.5 <= #330.out 16
	#347 toNextStartOsmos1timer <= #330.out 17
	#348 toNextStartOsmos2timer <= #330.out 18
	#349 statWordOsmos.6 <= #330.out 19
	#350 statWordOsmos.7 <= #330.out 20
END_MACRO
#351 MACRO сбор всех аварий и передача в панель(pin 1 "авария низкое давление РТ03.01/01": #231.out 1, pin 2 "авария низкое давление РТ03.01/02": #231.out 2)
	(* reserve *)
	(* авария доз.насоса Н03.04/02, 1=авария *)
	(* общая авария оборудования резервного осмоса *)
	(* авария клапанов 15-17, 1=авария *)
	(* общая авария оборудования основного осмоса *)
	(* авария доз.насоса Н03.04/01, 1=авария *)
	(* авария клапанов 12-14, 1=авария *)
	(* авария основного осмоса из / блока управления пусками *)
	(* авария резервного осмоса из / блока управлени пусками *)
	(* *авария основного осмоса по макс давлению датчика РТ03.03/01 *)
	(* *авария основного осмоса по макс давлению датчика РТ03.04/01 *)
	(* PSW336 *)
	(* авария насоса Р03.02/01 *)
	(* авария насоса Р03.02/02 *)
	(* ошибка блока дозирования Р03.02 *)
	(* авария доз.насоса Н03.04/01, 1=авария *)
	(* авария клапанов 12-14, 1=авария *)
	(* авария доз.насоса Н03.04/02, 1=авария *)
	(* авария клапанов 15-17, 1=авария *)
	(* *авария основного осмоса по макс давлению датчика РТ03.03/02 *)
	(* *авария основного осмоса по макс давлению датчика РТ03.04/02 *)
	(* авария клапана 18, 1=авария *)
	(* PSW337 *)
	#352 PANalarms.0 <= pin 1
	#353 PANalarms.1 <= pin 2
	#354 OR(DD1_DI_11, DD1_DI_7, PT030101alarm, PT030201alarm, PT030301alarm, PT030401alarm, QIT030101alarm, FIT030201alarm, FIT030301alarm, P030601alarm)
	#355 osmos1EquipmentAlarm <= #354
	#356 OR(#354, statWordOsmos.6)
	#357 OR(DD1_DI_12, DD1_DI_8, osmos2sensorsAlarm, P030602alarm)
	#358 osmos2EquipmentAlarm <= #357
	#359 OR(statWordOsmos.7, #357)
	#360 AND(#356, #359)
	#361 osmosTotalAlarm <= #360
	#362 PANalarms.2 <= statWordP0302.6
	#363 PANalarms.3 <= statWordP0302.7
	#364 PANalarms.4 <= DD1_DI_7
	#365 PANalarms.5 <= DD1_DI_8
	#366 PANalarms.6 <= P030601alarm
	#367 PANalarms.7 <= P030602alarm
	#368 PANalarms.8 <= DD1_DI_11
	#369 PANalarms.9 <= DD1_DI_12
	#370 PANalarms.10 <= DD1_DI_13
	#371 PANalarms.11 <= dosingErrorP0302
	#372 PANalarms.12 <= osmos1AlarmPT030301
	#373 PANalarms.13 <= osmos1AlarmPT030401
	#374 PANalarms.14 <= osmos2AlarmPT030302
	#375 PANalarms.15 <= osmos2AlarmPT030402
	#376 PANalarms.16 <= FIT0301alarm
	#377 PANalarms.17 <= PT030101alarm
	#378 PANalarms.18 <= PT030201alarm
	#379 PANalarms.19 <= PT030301alarm
	#380 PANalarms.20 <= PT030401alarm
	#381 PANalarms.21 <= QIT030101alarm
	#382 PANalarms.22 <= FIT030201alarm
	#383 PANalarms.23 <= FIT030301alarm
	#384 PANalarms.24 <= PT030102alarm
	#385 PANalarms.25 <= PT030202alarm
	#386 PANalarms.26 <= PT030302alarm
	#387 PANalarms.27 <= PT030402alarm
	#388 PANalarms.28 <= QIT030102alarm
	#389 PANalarms.29 <= FIT030202alarm
	#390 PANalarms.30 <= FIT030302alarm
	#391 PANalarms.31 <= LT0301alarm
END_MACRO
#392 MACRO настройки и состояние емкости V0207()
	(* низкий уровень в емкости V02.07  1 = true *)
	(* высокий уровень в емкости V02.07  1 = true *)
	#393 MOVE(EN: PAN_valuesActivator.6, PAN_V0207minHeight)
	#394 V0207minHeight <= #393
	#395 MOVE(EN: PAN_valuesActivator.6, PAN_V0207maxHeight)
	#396 V0207maxHeight <= #395
	#397 PAN_currentValue_V0207minHeight <= V0207minHeight
	#398 PAN_currentValue_V0207maxHeight <= V0207maxHeight
	#399 PAN_currentValue_V0207height <= LT0302realValue
	#400 >=(LT0302realValue, V0207maxHeight)
	#401 highLevelV0207 <= #400
	#402 <=(LT0302realValue, V0207minHeight)
	#403 lowLevelV0207 <= #402
END_MACRO
#404 WORD_TO_BOOL(PANsetWordOsmos)
#405 tof5:TOF(IN: #404, PT: T#1s)
#406 MOVE(EN: #405.Q, PANsetWordOsmos)
#407 setWordOsmos <= #406
#408 WORD_TO_BOOL(OPANsetWordOsmos)
#409 tof6:TOF(IN: #408, PT: T#1s)
#410 OR(#405.Q, #409.Q)
#411 MOVE(EN: #410, statWordOsmos)
#412 setWordOsmosOnStart <= #411
#413 MOVE(EN: #409.Q, OPANsetWordOsmos)
#414 setWordOsmos <= #413
#415 MACRO обработка аналоговых сигналов датчиков основного осмоса()
	(* сигнал датчика LT02.03 / уровень емкости V02.07 *)
	#416 controlAIpt030101:ControlAI(DD1_AI_2, -, PT030101maxValue)
	#417 PT030101realValue <= #416.out 1
	#418 PT030101alarm <= #416.out 2
	#419 controlAILT0203:ControlAI(DD1_AI_1, -, LT0203maxValue)
	#420 LT0302realValue <= #419.out 1
	#421 LT0301alarm <= #419.out 2
	#422 controlAIpt030201:ControlAI(DD1_AI_3, -, PT030201maxValue)
	#423 PT030201realValue <= #422.out 1
	#424 PT030201alarm <= #422.out 2
	#425 controlAIpt030301:ControlAI(DD1_AI_4, -, PT030301maxValue)
	#426 PT030301realValue <= #425.out 1
	#427 PT030301alarm <= #425.out 2
	#428 controlAIpt030401:ControlAI(DD1_AI_5, -, PT030401maxValue)
	#429 PT030401realValue <= #428.out 1
	#430 PT030401alarm <= #428.out 2
	#431 controlAIqit030101:ControlAI(DD1_AI_6, -, QIT030101maxValue)
	#432 QIT030101realValue <= #431.out 1
	#433 QIT030101alarm <= #431.out 2
	#434 controlAIfit030201:ControlAI(DD1_AI_7, -, FIT030201maxValue)
	#435 FIT030201realValue <= #434.out 1
	#436 FIT030201alarm <= #434.out 2
	#437 controlAIfit030301:ControlAI(DD1_AI_8, -, FIT030301maxValue)
	#438 FIT030301realValue <= #437.out 1
	#439 FIT030301alarm <= #437.out 2
END_MACRO
#440 MACRO передача показаний датчиков в панель оператора()
	#441 PAN_FIT0301realValue <= FIT0301realValue
	#442 PAN_PT030101realValue <= PT030101realValue
	#443 PAN_PT030201realValue <= PT030201realValue
	#444 PAN_PT030301realValue <= PT030301realValue
	#445 PAN_FIT030301realValue <= FIT030301realValue
	#446 PAN_PT030102realValue <= PT030102realValue
	#447 PAN_PT030202realValue <= PT030202realValue
	#448 PAN_PT030302realValue <= PT030302realValue
	#449 PAN_FIT030302realValue <= FIT030302realValue
	#450 PAN_PT030401realValue <= PT030401realValue
	#451 PAN_FIT030201realValue <= FIT030201realValue
	#452 PAN_QIT030101realValue <= QIT030101realValue
	#453 PAN_PT030402realValue <= PT030402realValue
	#454 PAN_FIT030202realValue <= FIT030202realValue
	#455 PAN_QIT030102realValue <= QIT030102realValue
END_MACRO
#456 MACRO передача на главный экран панели статусов работы()
	(* valve 18 *)
	(* valve 17 *)
	(* valve 16 *)
	(* valve 15 *)
	(* valve 14 *)
	(* valve 13 *)
	(* valve 12 *)
	(* P03.04/02 *)
	(* P03.04/01 *)
	#457 PANmainViewBools.2 <= DD1_DO_4
	#458 PANmainViewBools.3 <= DD1_DO_5
	#459 PANmainViewBools.4 <= P030601start
	#460 PANmainViewBools.5 <= P030602start
	#461 PANmainViewBools.6 <= DD1_DO_6
	#462 PANmainViewBools.7 <= DD1_DO_7
	#463 PANmainViewBools.8 <= DD1_DO_8
	#464 PANmainViewBools.9 <= DD1_DO_9
	#465 PANmainViewBools.10 <= DD1_DO_10
	#466 PANmainViewBools.11 <= DD1_DO_11
	#467 PANmainViewBools.12 <= DD1_DO_1
	#468 PANmainViewBools.13 <= NOT highLevelV0207
	#469 PANmainViewBools.14 <= NOT highLevelV0601
END_MACRO
#470 MACRO обмен сигналами с DD2 (ПР102) и обработка аналоговых сигналов рез.осмоса()
	(* передача производительности / Р03.06/02 через модбас *)
	(* производительность доз.насоса Р03.06/02 / в процентах 0...100% *)
	(* 5430 - это число, соответствующее 100% / производительности ЧРП (50Гц) / так показали эксперименты в Казани / по РЭ и обучающим видео Овна 50Гц / соответствует число 16384 / Не знаю кому верить / Это число надо уточнить при ПНР... *)
	(* передача производительности / Р03.06/01 через модбас *)
	(* производительность доз.насоса Р03.06/01 / в процентах 0...100% *)
	(* сигнал на запуск Р03.06/02 *)
	(* получить из DD2 *)
	(* авария насоса Р03.06/02 *)
	(* передать в DD2 *)
	(* сигнал на запуск Р03.06/01 *)
	(* авария насоса Р03.06/01 *)
	(* есть авария хотя бы одного датчика в резеврном осмосе / получить из DD2 (ПР102), 1=авария *)
	(* сигнал на старт Р03.01/02 *)
	(* сигнал на старт Р03.01/01 *)
	#471 DO_bit_mask_DD2.0 <= statWordP0301.4
	#472 P030601alarm <= stat_word_P030601_PLC.3
	#473 DO_bit_mask_DD2.1 <= statWordP0301.5
	#474 P030602alarm <= stat_word_P030602_PLC.3
	#475 MACRO командное слово Р03.06/01(pin 1 "пуск/стоп": P030601start)
		(* не используется *)
		(* 0=набор 1, 1=набор 2 *)
		(* не используется *)
		(* 0=реле 1 выключено, 1=реле 1 включено *)
		(* 0=данные недействительны, 1=данные действительны *)
		(* 0=изменение скорости1 (согласно 3-4), 1=изменение скорости 2 (согласно 3-5) *)
		(* 0=работа по заданию, 1=фиксированная частота(параметр 3-11) *)
		(* 0=нет сброса, 1=сброс *)
		(* 0=останов с замедлением, 1=пуск *)
		(* фиксация частоты, 0=есть, 1=нет *)
		(* быстрый останов, 0=есть, 1=нет *)
		(* останов выбегом, 0=есть, 1=нет *)
		(* торможение постоянным током, 0=есть, 1=нет. *)
		(* предустановленное значение, старший бит, 0=0, 1=1 *)
		(* предустановленное значение, младший бит, 0=0, 1=1 *)
		#476 com_word_P030601_PLC.0 <= 0
		#477 com_word_P030601_PLC.1 <= 0
		#478 com_word_P030601_PLC.2 <= 1
		#479 com_word_P030601_PLC.3 <= pin 1
		#480 com_word_P030601_PLC.6 <= pin 1
		#481 com_word_P030601_PLC.4 <= 1
		#482 com_word_P030601_PLC.5 <= 1
		#483 com_word_P030601_PLC.7 <= 0
		#484 com_word_P030601_PLC.8 <= 0
		#485 com_word_P030601_PLC.9 <= 0
		#486 com_word_P030601_PLC.10 <= 1
		#487 com_word_P030601_PLC.11 <= 0
		#488 com_word_P030601_PLC.12 <= 0
		#489 com_word_P030601_PLC.13 <= 0
		#490 com_word_P030601_PLC.14 <= 0
	END_MACRO
	#491 MACRO командное слово Р03.06/02(pin 1 "пуск/стоп": P030602start)
		(* не используется *)
		(* 0=набор 1, 1=набор 2 *)
		(* не используется *)
		(* 0=реле 1 выключено, 1=реле 1 включено *)
		(* 0=данные недействительны, 1=данные действительны *)
		(* 0=изменение скорости1 (согласно 3-4), 1=изменение скорости 2 (согласно 3-5) *)
		(* 0=работа по заданию, 1=фиксированная частота(параметр 3-11) *)
		(* 0=нет сброса, 1=сброс *)
		(* 0=останов с замедлением, 1=пуск *)
		(* фиксация частоты, 0=есть, 1=нет *)
		(* быстрый останов, 0=есть, 1=нет *)
		(* останов выбегом, 0=есть, 1=нет *)
		(* торможение постоянным током, 0=есть, 1=нет. *)
		(* предустановленное значение, старший бит, 0=0, 1=1 *)
		(* предустановленное значение, младший бит, 0=0, 1=1 *)
		#492 com_word_P030602_PLC.0 <= 0
		#493 com_word_P030602_PLC.1 <= 0
		#494 com_word_P030602_PLC.2 <= 1
		#495 com_word_P030602_PLC.3 <= pin 1
		#496 com_word_P030602_PLC.6 <= pin 1
		#497 com_word_P030602_PLC.4 <= 1
		#498 com_word_P030602_PLC.5 <= 1
		#499 com_word_P030602_PLC.7 <= 0
		#500 com_word_P030602_PLC.8 <= 0
		#501 com_word_P030602_PLC.9 <= 0
		#502 com_word_P030602_PLC.10 <= 1
		#503 com_word_P030602_PLC.11 <= 0
		#504 com_word_P030602_PLC.12 <= 0
		#505 com_word_P030602_PLC.13 <= 0
		#506 com_word_P030602_PLC.14 <= 0
	END_MACRO
	#507 WORD_TO_BOOL(DI_bit_mask_DD2)
	#508 osmos2sensorsAlarm <= #507
	#509 freqP030601:LIN_TRAFO(IN: Yout_Total_P030601, IN_MIN: 0, IN_MAX: 100, OUT_MIN: 0, OUT_MAX: 16384)
	#510 REAL_TO_WORD(#509.OUT)
	#511 set_freq_P030601_PLC <= #510
	#512 MACRO сигналы DD2 (ПР102)()
		(* давление датчик РТ03.01/02 *)
		(* давление датчик РТ03.02/02 *)
		(* давление датчик РТ03.03/02 *)
		(* давление датчик РТ03.04/02 *)
		(* расходомер FIT03.03/02 *)
		(* расходомер FIT03.02/02 *)
		(* кондуктомер QIT03.01/02 *)
		#513 fit030202:ControlAI(FIT030202rawValue, -, FIT030202maxValue)
		#514 FIT030202realValue <= #513.out 1
		#515 FIT030202alarm <= #513.out 2
		#516 pt030102:ControlAI(PT030102rawValue, -, PT030102maxValue)
		#517 PT030102realValue <= #516.out 1
		#518 PT030102alarm <= #516.out 2
		#519 fit030302:ControlAI(FIT030302rawValue, -, FIT030302maxValue)
		#520 FIT030302realValue <= #519.out 1
		#521 FIT030302alarm <= #519.out 2
		#522 pt030202:ControlAI(PT030202rawValue, -, PT030202maxValue)
		#523 PT030202realValue <= #522.out 1
		#524 PT030202alarm <= #522.out 2
		#525 qit030102:ControlAI(QIT030102rawValue, -, QIT030102maxValue)
		#526 QIT030102realValue <= #525.out 1
		#527 QIT030102alarm <= #525.out 2
		#528 pt030302:ControlAI(PT030302rawValue, -, PT030302maxValue)
		#529 PT030302realValue <= #528.out 1
		#530 PT030302alarm <= #528.out 2
		#531 pt030402:ControlAI(PT030402rawValue, -, PT030402maxValue)
		#532 PT030402realValue <= #531.out 1
		#533 PT030402alarm <= #531.out 2
	END_MACRO
	#534 freqP030602:LIN_TRAFO(IN: Yout_Total_P030602, IN_MIN: 0, IN_MAX: 100, OUT_MIN: 0, OUT_MAX: 16384)
	#535 REAL_TO_WORD(#534.OUT)
	#536 set_freq_P030602_PLC <= #535
END_MACRO
#537 MACRO передача в панель состояния и наработки осмосов()
	#538 PANstatWordOsmos <= statWordOsmos
	#539 PANdaysOfWorkOsmos1 <= daysOfWorkOsmos1
	#540 PANhoursOfWorkOsmos1 <= hoursOfWorkOsmos1
	#541 PANminutesOfWorkOsmos1 <= minutesOfWorkOsmos1
	#542 PANsecondsOfWorkOsmos1 <= secondsOfWorkOsmos1
	#543 PANtoNextStartOsmos1timer <= toNextStartOsmos1timer
	#544 PANcounterOsmos1 <= counterOsmos1
	#545 PANcounterOsmos2 <= counterOsmos2
	#546 PANdaysOfWorkOsmos2 <= daysOfWorkOsmos2
	#547 PANhoursOfWorkOsmos2 <= hoursOfWorkOsmos2
	#548 PANminutesOfWorkOsmos2 <= minutesOfWorkOsmos2
	#549 PANsecondsOfWorkOsmos2 <= secondsOfWorkOsmos2
	#550 PANtoNextStartOsmos2timer <= toNextStartOsmos2timer
END_MACRO
#551 MACRO передача наработки и состояния доз.насоса Р03.02 в панель()
	#552 PANstatWordP0302 <= statWordP0302
	#553 PANdaysOfWorkP030201 <= daysOfWorkP030201
	#554 PANhoursOfWorkP030201 <= hoursOfWorkP030201
	#555 PANminutesOfWorkP030201 <= minutesOfWorkP030201
	#556 PANsecondsOfWorkP030201 <= secondsOfWorkP030201
	#557 PANtoNextStartP030201timer <= toNextStartP030201timer
	#558 PANcounterP030201 <= counterP030201
	#559 PANdaysOfWorkP030202 <= daysOfWorkP030202
	#560 PANhoursOfWorkP030202 <= hoursOfWorkP030202
	#561 PANminutesOfWorkP030202 <= minutesOfWorkP030202
	#562 PANsecondsOfWorkP030202 <= secondsOfWorkP030202
	#563 PANtoNextStartP030202timer <= toNextStartP030202timer
	#564 PANcounterP030202 <= counterP030202
END_MACRO
_END_CFC_
END_PROGRAM
